(* IEC 61131-3 sources: LASAL/Class/MoveController, 1 file *)

(* ---- MoveController.st ---- *)
(*!
<Class
	Name               = "MoveController"
	Revision           = "0.0"
	RealtimeTask       = "true"
	DefRealtime        = "1 ms"
	CyclicTask         = "false"
	BackgroundTask     = "false"
	Sigmatek           = "false"
	OSInterface        = "false"
	HighPriority       = "false"
	Automatic          = "false"
	UpdateMode         = "Prescan"
	SharedCommandTable = "true"
	Objectsize         = "(600,480)">
	<Channels>
		<Server Name="P_currentloop" Visualized="false" Initialize="false" WriteProtected="false" Retentive="File"/>
		<Server Name="sPower" Visualized="false" Initialize="false" WriteProtected="false" Retentive="false"/>
		<Server Name="State" Visualized="false" Initialize="false" WriteProtected="false" Retentive="false"/>
		<Server Name="Status" Visualized="false" Initialize="false" WriteProtected="false" Retentive="false"/>
		<Server Name="Z_currentTarget" Visualized="false" Initialize="false" WriteProtected="false" Retentive="File"/>
		<Server Name="Z_DownPos" Visualized="false" Initialize="false" WriteProtected="false" Retentive="File"/>
		<Server Name="Z_positiontarget" Visualized="false" Initialize="false" WriteProtected="false" Retentive="false"/>
		<Client Name="CommandServer" Required="true" Internal="false"/>
		<Client Name="lmcX" Required="true" Internal="false"/>
		<Client Name="lmcY" Required="true" Internal="false"/>
		<Client Name="lmcYShort" Required="true" Internal="false"/>
		<Client Name="lmcZ" Required="true" Internal="false"/>
		<Client Name="ResetDummy" Required="true" Internal="false"/>
		<Client Name="Z_current" Required="true" Internal="false"/>
	</Channels>
</Class>
*)
MoveController : CLASS
	TYPE
	  _MotionState :  //! <Type Public="true" Name="_MotionState"/>
	  (
	    _Safe,
	    _Homing,
	    _InHomepos,
	    _EnableShort,
	    _HomeShort,
	    _InPosHomeShort,
	    _Waiting,
	    _MovingAbsolute,
	    _moveready,
	    _MovingRelative,
	    _Pick,
	    _Place,
	    _Error
	  )$UDINT;
#pragma pack(push, 1)
	  _Move : STRUCT
	    Start : DINT;
	    X : DINT;
	    Z : DINT;
	    Y : DINT;
	    Speed : DINT;
	    Acc : DINT;
	    YSpeed : DINT;
	    YAcc : DINT;
	  END_STRUCT;
#pragma pack(pop)
	  _Status :  //! <Type Public="true" Name="_Status"/>
	  (
	    _Idle,
	    _PowerOn,
	    _PowerIsOn,
	    _refRun,
	    _RefrunOk,
	    _MoveAbosolute,
	    _InPosition
	  )$UDINT;
	  _Z_stepper :
	  (
	    __Idle,
	    __MoveDown,
	    __Currentloop,
	    __MoveUp
	  )$UDINT;
	END_TYPE
  //Servers:
	Status 	: SvrChCmd__Status_PTofCls_MoveController;
	sPower 	: SvrCh_DINT;
	State 	: SvrCh__MotionState_PTofCls_MoveController;
	Z_positiontarget 	: SvrCh_DINT;
	Z_currentTarget 	: SvrCh_DINT;
	Z_DownPos 	: SvrCh_DINT;
	P_currentloop 	: SvrCh_REAL;
  //Clients:
	lmcX 	: CltChCmd__LMCAxis;
	lmcY 	: CltChCmd__LMCAxis;
	ResetDummy 	: CltCh_DINT;
	CommandServer 	: CltChCmd_CommandServer;
	lmcYShort 	: CltChCmd__LMCAxis;
	lmcZ 	: CltChCmd__LMCAxis;
	Z_current 	: CltCh_DINT;
  //Variables:
		NewMove 	: _Move;
		IsMoving 	: BOOL;
		Z_stepper 	: _Z_stepper;
		DeltaCurrent 	: REAL;
  //Functions:

	FUNCTION VIRTUAL GLOBAL Init;

	FUNCTION VIRTUAL GLOBAL RtWork
		VAR_INPUT
			EAX 	: UDINT;
		END_VAR
		VAR_OUTPUT
			state (EAX) 	: UDINT;
		END_VAR;

	FUNCTION GLOBAL MoveAxis
		VAR_INPUT
			XPos 	: DINT;
			YPos 	: DINT;
			Speed 	: DINT;
			Accel 	: DINT;
			YSpeed 	: DINT;
			YAcc 	: DINT;
		END_VAR;

	FUNCTION GLOBAL TogglePower
		VAR_INPUT
			Power 	: BOOL;
		END_VAR;

	FUNCTION StateMachine;

	FUNCTION Z_control_loop;
  //Tables:
	FUNCTION @STD
		VAR_OUTPUT
			ret_code	: CONFSTATES;
		END_VAR;
	FUNCTION GLOBAL TAB @CT_;
END_CLASS;

#pragma usingLtd _LMCAxis
#pragma usingLtd CommandServer

FUNCTION VIRTUAL GLOBAL MoveController::Init
END_FUNCTION

FUNCTION VIRTUAL GLOBAL MoveController::RtWork
	VAR_INPUT
		EAX 	: UDINT;
	END_VAR
	VAR_OUTPUT
		state (EAX) 	: UDINT;
	END_VAR

  StateMachine();
  Z_control_loop();
	state := READY;
END_FUNCTION

FUNCTION MoveController::StateMachine

case State of

_MotionState::_Safe:
  IF sPower THEN
    IF lmcX.AxisStatus.ReadyToPowerOn & lmcY.AxisStatus.ReadyToPowerOn THEN
      lmcX.PowerOn(Mode:=::_LMCAXIS_MOVEDIRECTION::LMCAXIS_MOVE_ANY_WAY);
      lmcY.PowerOn(Mode:=::_LMCAXIS_MOVEDIRECTION::LMCAXIS_MOVE_ANY_WAY);
      //lmcz.PowerOn(Mode:=::_LMCAXIS_MOVEDIRECTION::LMCAXIS_MOVE_ANY_WAY);
      State := _MotionState::_Homing;
    END_IF;
  END_IF;

_MotionState::_Homing:
  IF lmcX.AxisStatus.PowerOn THEN
    lmcX.MoveReference(Mode:=_LMCAXIS_REFMODE.NoZImpulse , Position:=0, VRef1:=200000, VRef2:=50000, Accel:=5000000, PositionWindow:=5000, RefJerk:=0);
    lmcY.MoveReference(Mode:=_LMCAXIS_REFMODE.NoZImpulse , Position:=0, VRef1:=2000000, VRef2:=500000, Accel:=20000000, PositionWindow:=5000, RefJerk:=0);
    //lmcz.MoveReference(Mode:=_LMCAXIS_REFMODE.NoZImpulse or _LMCAXIS_REFMODE.RefDirection, Position:=0, VRef1:=2000000, VRef2:=500000, Accel:=20000000, PositionWindow:=5000, RefJerk:=0);
    State:=_MotionState::_InHomepos;
  end_if;
  //lmcY.MoveReference(Mode:=_LMCAXIS_REFMODE.NoZImpulse |_LMCAXIS_REFMODE.RefDirection , Position:=, VRef1:=, VRef2:=, Accel:=, PositionWindow:=, RefJerk:=);

_MotionState::_InHomepos:
  IF lmcX.AxisStatus.IsReferenced & lmcY.AxisStatus.IsReferenced THEN
    CommandServer.SendStatus(Status:=1); //delete if short stroke is implemented again
    //lmcZ.CoupleUserPos(MaxVel:=lmcZ.VMax, MaxAcc:=lmcz.AMax, pMasterPos:=#Z_positiontarget, DeltaPos:=0, GearMul:=100, GearDiv:=100, Mode:=::_LMCAXIS_COUPLE_GEAR_MODE::LMCAXIS_COUPLE_PROFILE_NO_GEAR, MaxJerk:=0);
    ResetDummy.Write(input:=0);
    State:=_MotionState::_Waiting;
  END_IF;

_MotionState::_EnableShort:
  lmcYShort.PowerOn(Mode:=::_LMCAXIS_MOVEDIRECTION::LMCAXIS_MOVE_ANY_WAY);
  State:=_MotionState::_HomeShort;

_MotionState::_HomeShort:
  IF lmcYShort.AxisStatus.PowerOn THEN
    lmcYShort.MoveReference(Mode:=_LMCAXIS_REFMODE.NoZImpulse , Position:=0, VRef1:=2000, VRef2:=1500, Accel:=1000, PositionWindow:=10000, RefJerk:=0);
  State := _MotionState::_InPosHomeShort;
  END_IF;

_MotionState::_InPosHomeShort:
  IF lmcYShort.AxisStatus.IsReferenced THEN
    CommandServer.SendStatus(Status:=1);
    State := _MotionState::_Waiting;
  END_IF;

_MotionState::_Waiting:
  IF lmcX.AxisStatus.PowerOn THEN
    IF NewMove.Start THEN
      State:=_MotionState::_MovingAbsolute;
    END_IF;
  END_IF;
  IF sPower = FALSE THEN
    lmcX.PowerOff(Mode:=::_LMCAXIS_POWER_OFF_MODE::LMCAXIS_SMOOTH_STOPP);
    lmcY.PowerOff(Mode:=::_LMCAXIS_POWER_OFF_MODE::LMCAXIS_SMOOTH_STOPP);
    State:=_MotionState::_Safe;
  END_IF;

_MotionState::_MovingAbsolute:
//  if NewMove.X> lmcX.SWMaxPos then
//  end_if;
    lmcx.MoveAbsolute(Position:=NewMove.X, Speed:=NewMove.Speed, Accel:=NewMove.Acc, Decel:=NewMove.Acc, Jerk:=0);
    lmcY.MoveAbsolute(Position:=NewMove.Y, Speed:=NewMove.YSpeed, Accel:=NewMove.YAcc, Decel:=NewMove.YAcc, Jerk:=0);
    State:=_MotionState::_moveready;

_MotionState::_moveready:
    IF lmcX.InPosition(Mode:=::_LMCAXIS_QUERY_POSITION_MODE::LMCAXIS_ACTPOS_IN_WINDOW_APP_UNITS, PositionWindow:=1000) &
     lmcY.InPosition(Mode:=::_LMCAXIS_QUERY_POSITION_MODE::LMCAXIS_ACTPOS_IN_WINDOW_APP_UNITS, PositionWindow:=1000) THEN
      NewMove.Start := FALSE;
      CommandServer.SendStatus(Status:=1);
      State:=_MotionState::_Waiting;
    END_IF;

END_CASE;

END_FUNCTION

FUNCTION MoveController::Z_control_loop
Z_current:=Z_current.Read();

if !! lmcZ.AxisStatus.IsReferenced | !! lmcZ.AxisStatus.PowerOn then
  Z_stepper:=_Z_stepper::__Idle;
end_if;

case Z_stepper of

_Z_stepper::__Idle:
  if lmcZ.AxisStatus.IsReferenced & lmcZ.AxisStatus.PowerOn then
    Z_stepper:=_Z_stepper::__MoveDown;
  end_if;

_Z_stepper::__MoveDown:
  if NewMove.Z then
    Z_positiontarget:=Z_DownPos;
    Z_stepper:=_Z_stepper::__Currentloop;
  end_if;

_Z_stepper::__Currentloop:

  //Cotrol loop, if current is higher then setpoint move a bit up.
  DeltaCurrent:=to_real(Z_currentTarget) - to_real(Z_current);
  Z_positiontarget+=to_dint(DeltaCurrent * P_currentloop);

  if NewMove.Z=false then
    Z_stepper:=_Z_stepper::__MoveUp;
  end_if;

_Z_stepper::__MoveUp:
  Z_positiontarget:=0;
  Z_stepper:=_Z_stepper::__MoveDown;

end_case;

END_FUNCTION

FUNCTION GLOBAL MoveController::MoveAxis
	VAR_INPUT
		XPos 	: DINT;
		YPos 	: DINT;
		Speed 	: DINT;
		Accel 	: DINT;
		YSpeed 	: DINT;
		YAcc 	: DINT;
	END_VAR

  NewMove.X := XPos;
  NewMove.Y := YPos;
  NewMove.Speed := Speed;
  NewMove.Acc := Accel;
  NewMove.YSpeed := YSpeed;
  NewMove.YAcc := YAcc;

  NewMove.Start:=TRUE;

END_FUNCTION

FUNCTION GLOBAL MoveController::TogglePower
	VAR_INPUT
		Power 	: BOOL;
	END_VAR
  sPower:=Power;

END_FUNCTION
